// TIA Portal project "3M - 2" (V16)

(* hardware
DEVICE "S7-1200 station_1"  S7-1200 Station
   slot 0: "Rack_0"  S7-1200 Rack  Rack  V1.0
   slot 1: "PLC_1"  CPU 1212C AC/DC/Rly  6ES7 212-1BE40-0XB0  V4.0
*)

// ===== PLC "PLC_1"  CPU 1212C AC/DC/Rly =====

VAR_GLOBAL   // PLC tag table "Default tag table"
   "K1" AT %Q0.0 : Bool;
   "stop1" AT %I0.4 : Bool;
   "k2" AT %Q0.1 : Bool;
   "X" AT %M0.2 : Bool;
   "K3" AT %Q0.2 : Bool;
   "start1" AT %I0.2 : Bool;
   "Tag_2" AT %M0.1 : Bool;
   "Tag_3" AT %M0.3 : Bool;
   "Tag_4" AT %M0.4 : Bool;
   "Tag_5" AT %M1.1 : Bool;
   "Tag_6" AT %M1.0 : Bool;
   "Tag_1" AT %M0.5 : Bool;
   "STOP" AT %I0.3 : Bool;
END_VAR

// folder: System blocks/Program resources

DATA_BLOCK "T4"   // DB1
{ S7_Optimized_Access := 'TRUE' }
AUTHOR : Simatic
FAMILY : IEC
NAME : IEC_TMR
VERSION : 1.0
// stored: InstanceOfName IEC_TIMER
"IEC_TIMER"
BEGIN
END_DATA_BLOCK

DATA_BLOCK "T1"   // DB2
{ S7_Optimized_Access := 'TRUE' }
AUTHOR : Simatic
FAMILY : IEC
NAME : IEC_TMR
VERSION : 1.0
// stored: InstanceOfName IEC_TIMER
"IEC_TIMER"
BEGIN
END_DATA_BLOCK

DATA_BLOCK "T2"   // DB3
{ S7_Optimized_Access := 'TRUE' }
AUTHOR : Simatic
FAMILY : IEC
NAME : IEC_TMR
VERSION : 1.0
// stored: InstanceOfName IEC_TIMER
"IEC_TIMER"
BEGIN
END_DATA_BLOCK

DATA_BLOCK "T3"   // DB4
{ S7_Optimized_Access := 'TRUE' }
AUTHOR : Simatic
FAMILY : IEC
NAME : IEC_TMR
VERSION : 1.0
// stored: InstanceOfName IEC_TIMER
"IEC_TIMER"
BEGIN
END_DATA_BLOCK

// folder: (top level)

ORGANIZATION_BLOCK "Main"   // OB1, LAD, ProgramCycle
TITLE = "Main Program Sweep (Cycle)"
{ S7_Optimized_Access := 'TRUE' }
VERSION : 0.1
   VAR_INPUT
      Initial_Call : Bool;   // Initial call of this OB
      Remanence : Bool;   // =True, if remanent data are available
   END_VAR
BEGIN

REGION Network 1: start
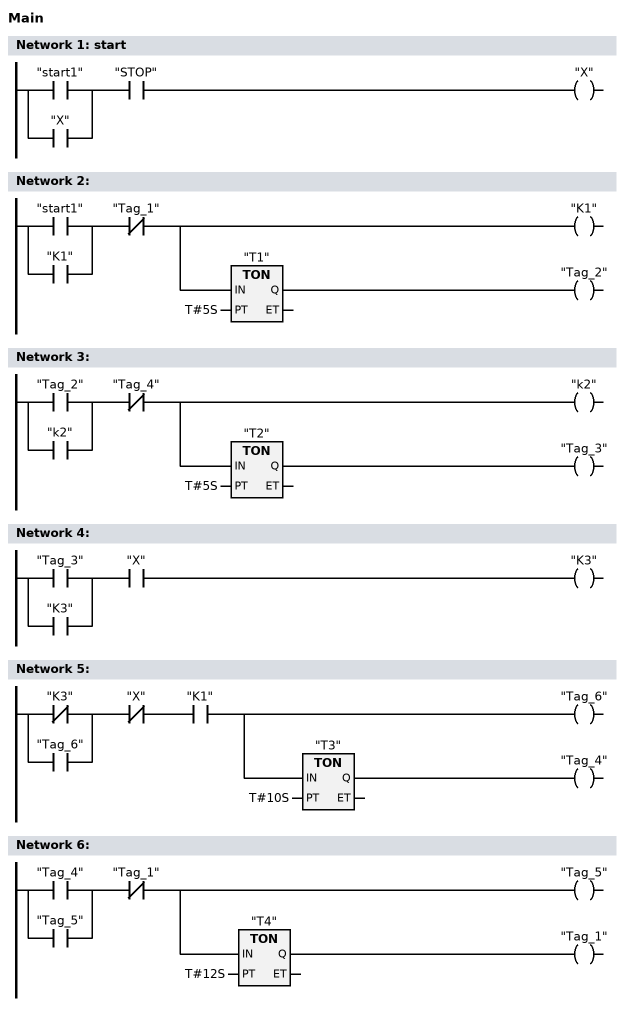
   RUNG wire#powerrail
      Contact( "start1" )
      wire#w1
      Contact( "STOP" )
      Coil( "X" )
   END_RUNG
   RUNG wire#powerrail
      Contact( "X" )
   END_RUNG wire#w1
   // the same network as SCL:
   "X" := ("start1" OR "X") AND "STOP";
END_REGION

REGION Network 2
   "K1" := ("start1" OR "K1") AND NOT "Tag_1";
   "T1".TON(IN := "K1", PT := T#5S);
   "Tag_2" := "T1".Q;
END_REGION

REGION Network 3
   "k2" := ("Tag_2" OR "k2") AND NOT "Tag_4";
   "T2".TON(IN := "k2", PT := T#5S);
   "Tag_3" := "T2".Q;
END_REGION

REGION Network 4
   RUNG wire#powerrail
      Contact( "Tag_3" )
      wire#w1
      Contact( "X" )
      Coil( "K3" )
   END_RUNG
   RUNG wire#powerrail
      Contact( "K3" )
   END_RUNG wire#w1
   // the same network as SCL:
   "K3" := ("Tag_3" OR "K3") AND "X";
END_REGION

REGION Network 5
   "Tag_6" := (NOT "K3" OR "Tag_6") AND NOT "X" AND "K1";
   "T3".TON(IN := "Tag_6", PT := T#10S);
   "Tag_4" := "T3".Q;
END_REGION

REGION Network 6
   "Tag_5" := ("Tag_4" OR "Tag_5") AND NOT "Tag_1";
   "T4".TON(IN := "Tag_5", PT := T#12S);
   "Tag_1" := "T4".Q;
END_REGION
END_ORGANIZATION_BLOCK